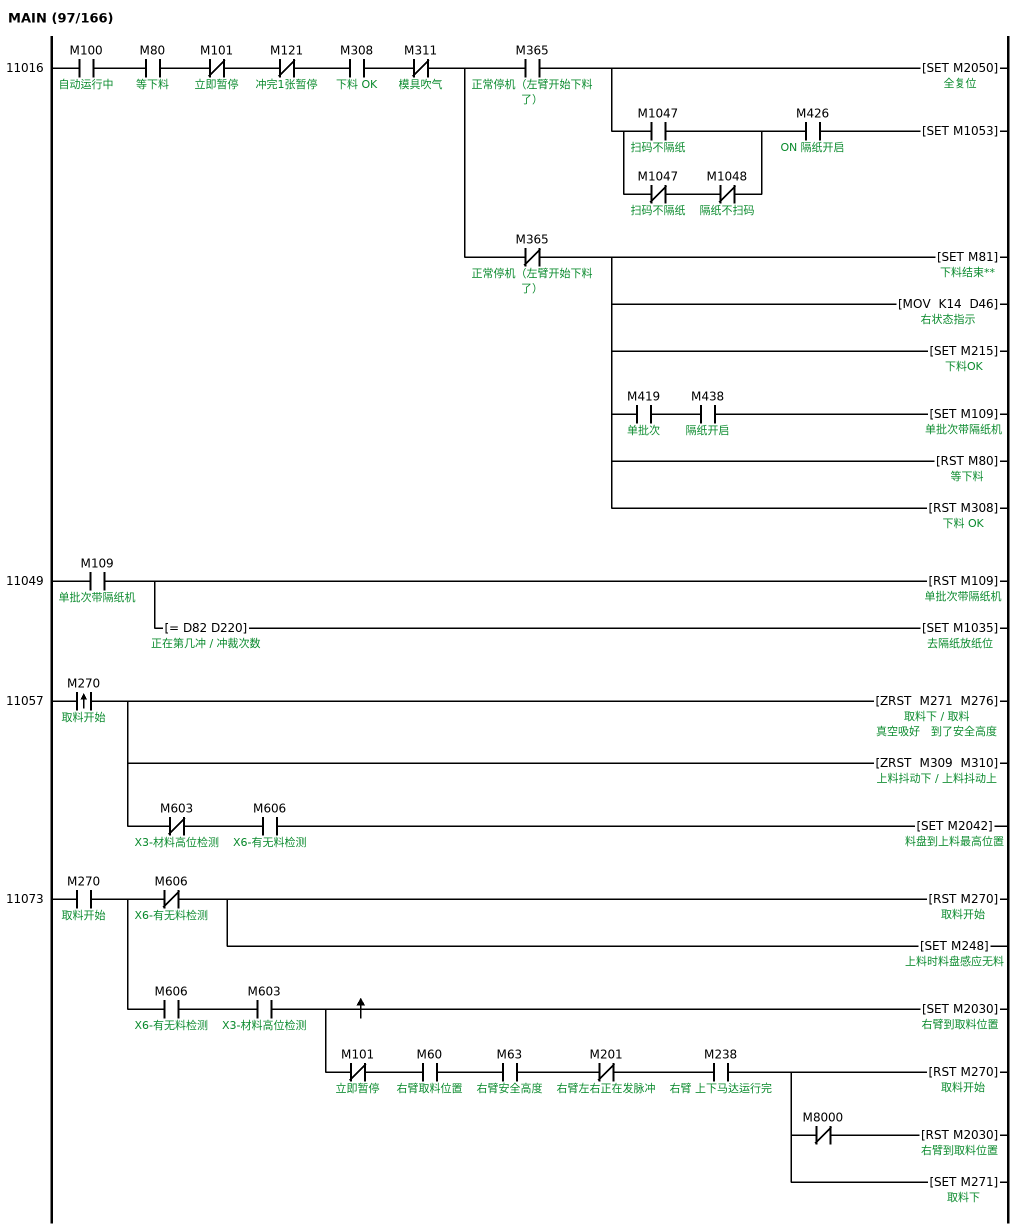
[picture p96: ladder of MAIN, rungs at steps 11016 to 11073]
11016 LD      M100  ; 自动运行中
      AND     M80  ; 等下料
      ANI     M101  ; 立即暂停
      ANI     M121  ; 冲完1张暂停
      AND     M308  ; 下料 OK
      ANI     M311  ; 模具吹气
      MPS
      AND     M365  ; 正常停机（左臂开始下料了）
      SET     M2050  ; 全复位
      LD      M1047  ; 扫码不隔纸
      LDI     M1047  ; 扫码不隔纸
      ANI     M1048  ; 隔纸不扫码
      ORB
      ANB
      AND     M426  ; ON 隔纸开启
      SET     M1053
      MPP
      ANI     M365  ; 正常停机（左臂开始下料了）
      SET     M81  ; 下料结束**
      MOV     K14 D46
      SET     M215  ; 下料OK
      MPS
      AND     M419  ; 单批次
      AND     M438  ; 隔纸开启
      SET     M109  ; 单批次带隔纸机
      MPP
      RST     M80  ; 等下料
      RST     M308  ; 下料 OK
11049 LD      M109  ; 单批次带隔纸机
      RST     M109  ; 单批次带隔纸机
      AND=    D82 D220  ; 正在第几冲 / 冲裁次数
      SET     M1035  ; 去隔纸放纸位
11057 LDP     M270  ; 取料开始
      ZRST    M271 M276  ; 取料下
        [note] M271亮，安全高度不动时，启动此行
      ZRST    M309 M310  ; 上料抖动下 / 上料抖动上
      ANI     M603  ; X3-材料高位检测
      AND     M606  ; X6-有无料检测
      SET     M2042  ; 料盘到上料最高位置
11073 LD      M270  ; 取料开始
      MPS
      ANI     M606  ; X6-有无料检测
      RST     M270  ; 取料开始
      SET     M248  ; 上料时料盘感应无料
      MPP
      AND     M606  ; X6-有无料检测
      AND     M603  ; X3-材料高位检测
      MPS
      MEP
      SET     M2030  ; 右臂到取料位置
      MPP
      ANI     M101  ; 立即暂停
      AND     M60  ; 右臂取料位置
      AND     M63  ; 右臂安全高度
      ANI     M201  ; 右臂左右正在发脉冲
      AND     M238  ; 右臂 上下马达运行完
      RST     M270  ; 取料开始
      MPS
      ANI     M8000
      RST     M2030  ; 右臂到取料位置
      MPP
      SET     M271  ; 取料下
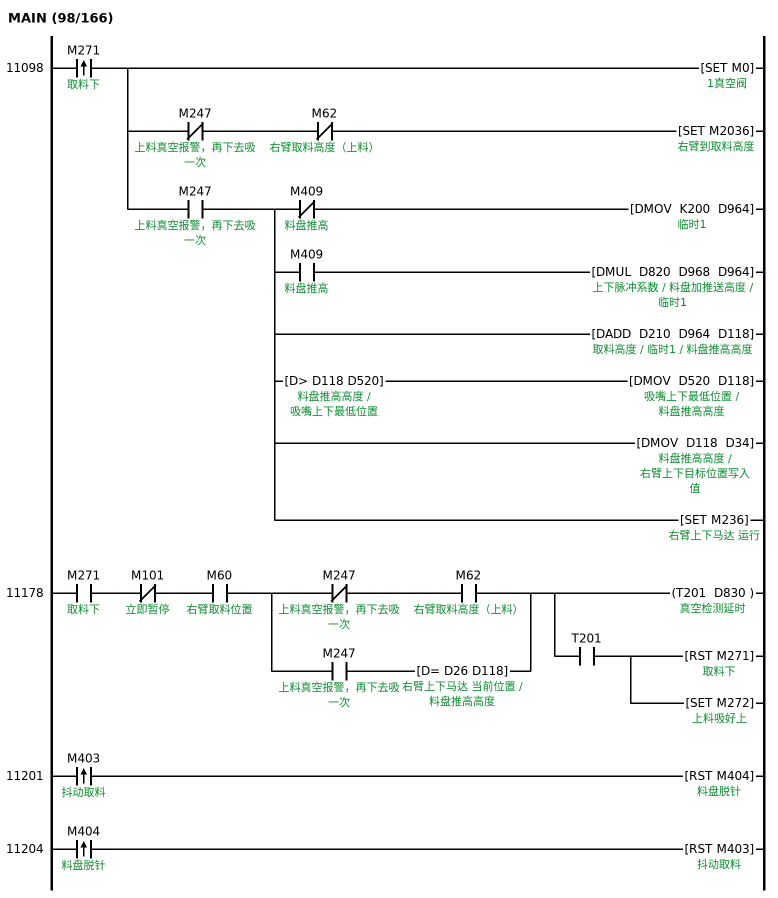
11098 LDP     M271  ; 取料下
      SET     M0  ; 1真空阀
      MPS
      ANI     M247  ; 上料真空报警，再下去吸一次
      ANI     M62  ; 右臂取料高度（上料）
      SET     M2036  ; 右臂到取料高度
      MPP
      AND     M247  ; 上料真空报警，再下去吸一次
      MPS
      ANI     M409  ; 料盘推高
      DMOV    K200 D964
      MRD
      AND     M409  ; 料盘推高
      DMUL    D820 D968 D964
      MPP
      DADD    D210 D964 D118  ; 料盘推高高度
      MPS
      ANDD>   D118 D520  ; 料盘推高高度 / 吸嘴上下最低位置
      DMOV    D520 D118
      MPP
      DMOV    D118 D34
      SET     M236  ; 右臂上下马达 运行
11178 LD      M271  ; 取料下
      ANI     M101  ; 立即暂停
      AND     M60  ; 右臂取料位置
      LDI     M247  ; 上料真空报警，再下去吸一次
      AND     M62  ; 右臂取料高度（上料）
      LD      M247  ; 上料真空报警，再下去吸一次
      ANDD=   D26 D118  ; 右臂上下马达 当前位置 / 料盘推高高度
      ORB
      ANB
      OUT     T201 D830  ; 真空检测延时
      AND     T201
      RST     M271  ; 取料下
      SET     M272  ; 上料吸好上
11201 LDP     M403  ; 抖动取料
      RST     M404  ; 料盘脱针
11204 LDP     M404  ; 料盘脱针
      RST     M403  ; 抖动取料
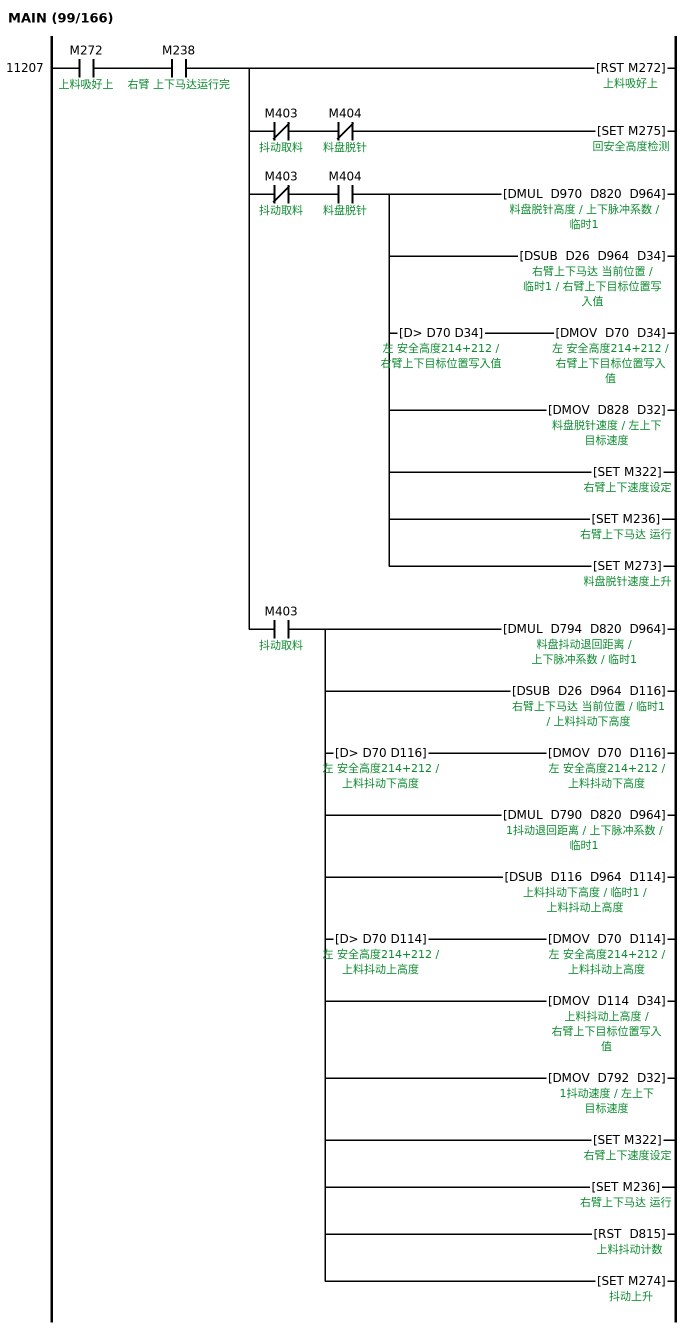
11207 LD      M272  ; 上料吸好上
      AND     M238  ; 右臂 上下马达运行完
      RST     M272  ; 上料吸好上
      MPS
      ANI     M403  ; 抖动取料
      ANI     M404  ; 料盘脱针
      SET     M275  ; 回安全高度检测
      MRD
      ANI     M403  ; 抖动取料
      AND     M404  ; 料盘脱针
      DMUL    D970 D820 D964  ; 料盘脱针高度
      DSUB    D26 D964 D34
      MPS
      ANDD>   D70 D34  ; 左 安全高度214+212 / 右臂上下目标位置写入值
      DMOV    D70 D34
      MPP
      DMOV    D828 D32  ; 左上下 目标速度
      SET     M322  ; 右臂上下速度设定
      SET     M236  ; 右臂上下马达 运行
      SET     M273  ; 料盘脱针速度上升
      MPP
      AND     M403  ; 抖动取料
      DMUL    D794 D820 D964
      DSUB    D26 D964 D116  ; 上料抖动下高度
      MPS
      ANDD>   D70 D116  ; 左 安全高度214+212 / 上料抖动下高度
      DMOV    D70 D116
      MPP
      DMUL    D790 D820 D964
      DSUB    D116 D964 D114  ; 上料抖动上高度
      MPS
      ANDD>   D70 D114  ; 左 安全高度214+212 / 上料抖动上高度
      DMOV    D70 D114
      MPP
      DMOV    D114 D34
      DMOV    D792 D32
      SET     M322  ; 右臂上下速度设定
      SET     M236  ; 右臂上下马达 运行
      RST     D815  ; 上料抖动计数
      SET     M274  ; 抖动上升
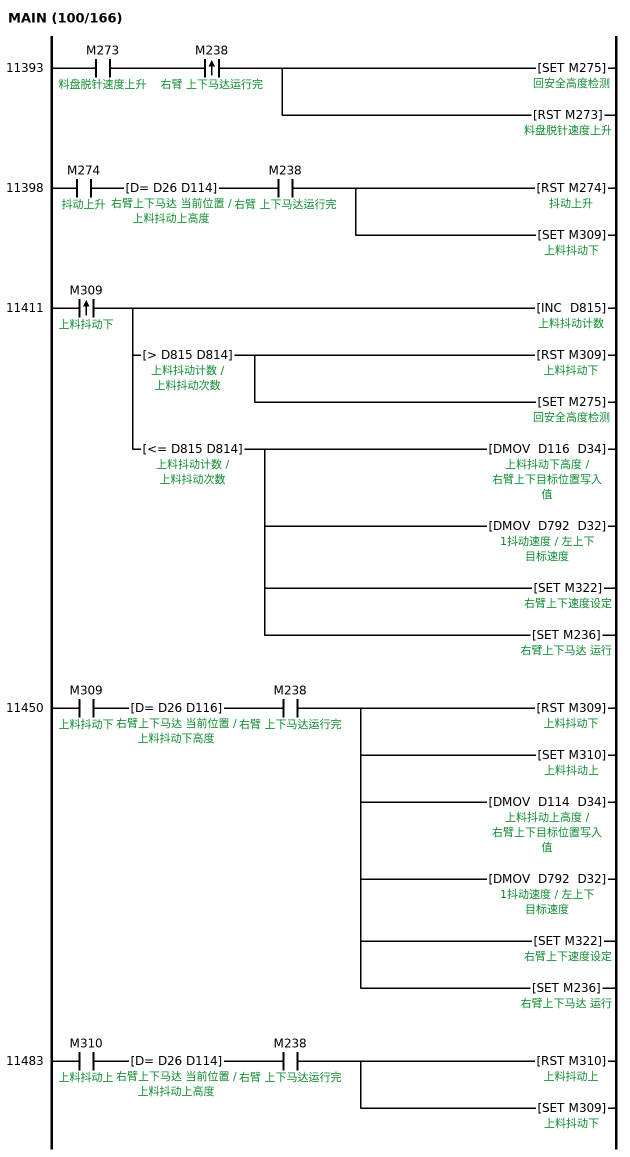
11393 LD      M273  ; 料盘脱针速度上升
      ANDP    M238  ; 右臂 上下马达运行完
      SET     M275  ; 回安全高度检测
      RST     M273  ; 料盘脱针速度上升
11398 LD      M274  ; 抖动上升
      ANDD=   D26 D114  ; 右臂上下马达 当前位置 / 上料抖动上高度
      AND     M238  ; 右臂 上下马达运行完
      RST     M274  ; 抖动上升
      SET     M309  ; 上料抖动下
11411 LDP     M309  ; 上料抖动下
      INC     D815
      MPS
      AND>    D815 D814  ; 上料抖动计数 / 上料抖动次数
      RST     M309  ; 上料抖动下
      SET     M275  ; 回安全高度检测
      MPP
      AND<=   D815 D814  ; 上料抖动计数 / 上料抖动次数
      DMOV    D116 D34
      DMOV    D792 D32
      SET     M322  ; 右臂上下速度设定
      SET     M236  ; 右臂上下马达 运行
11450 LD      M309  ; 上料抖动下
      ANDD=   D26 D116  ; 右臂上下马达 当前位置 / 上料抖动下高度
      AND     M238  ; 右臂 上下马达运行完
      RST     M309  ; 上料抖动下
      SET     M310  ; 上料抖动上
      DMOV    D114 D34
      DMOV    D792 D32
      SET     M322  ; 右臂上下速度设定
      SET     M236  ; 右臂上下马达 运行
11483 LD      M310  ; 上料抖动上
      ANDD=   D26 D114  ; 右臂上下马达 当前位置 / 上料抖动上高度
      AND     M238  ; 右臂 上下马达运行完
      RST     M310  ; 上料抖动上
      SET     M309  ; 上料抖动下
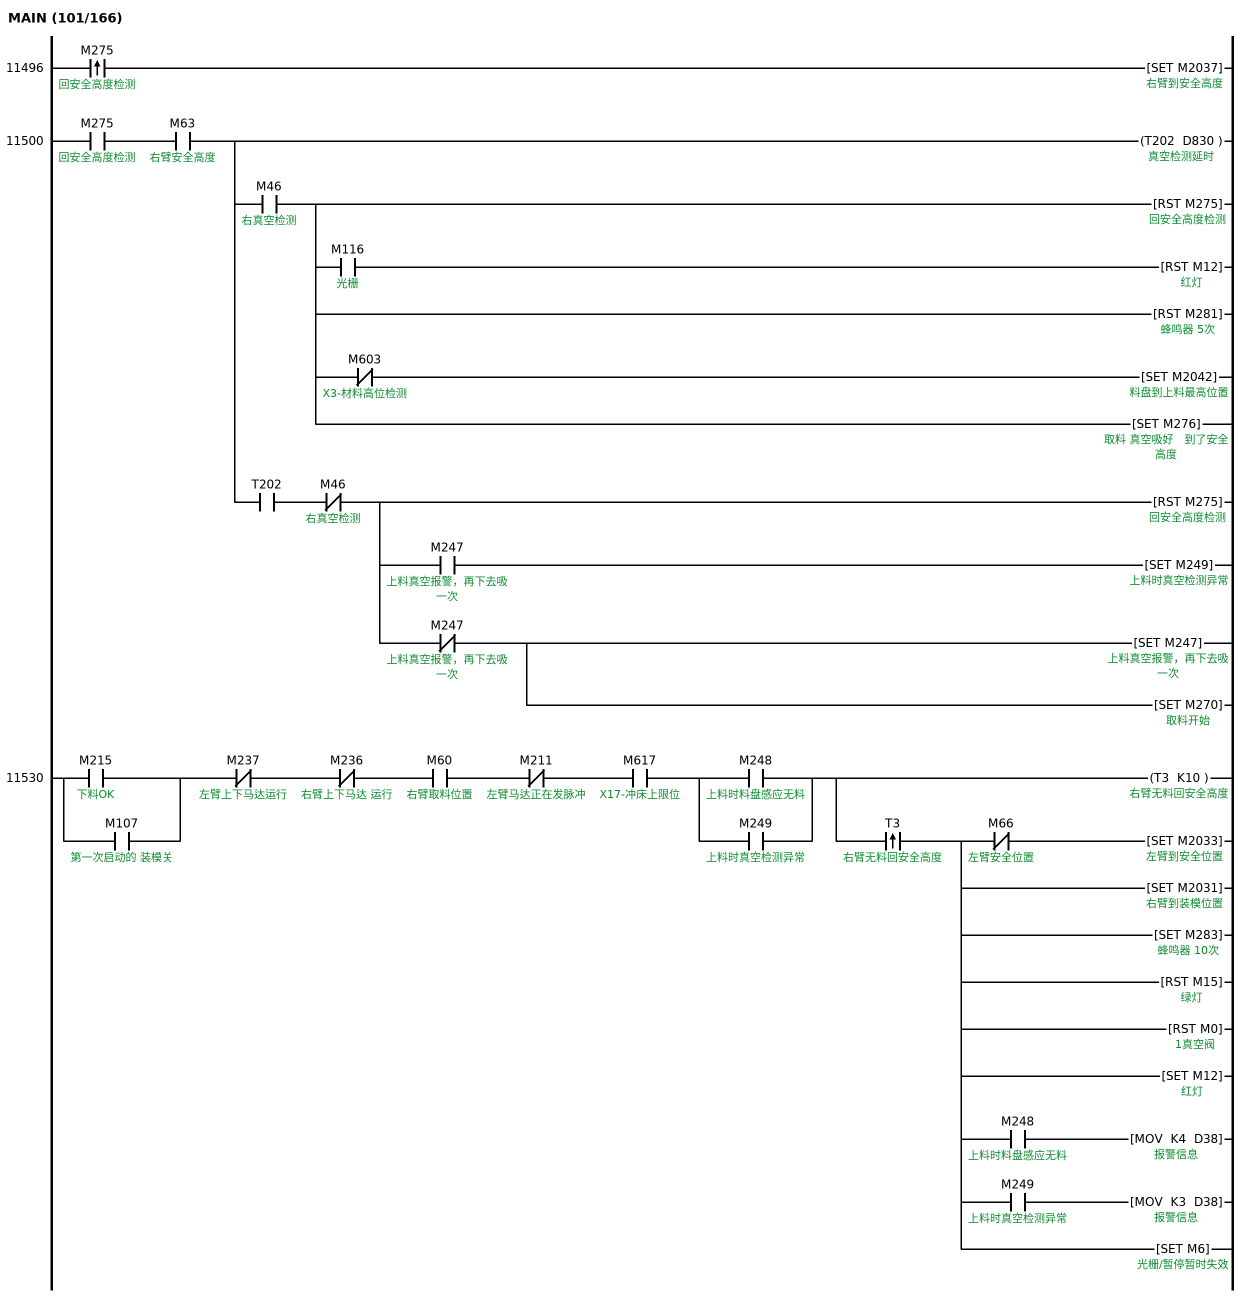
11496 LDP     M275  ; 回安全高度检测
      SET     M2037  ; 右臂到安全高度
11500 LD      M275  ; 回安全高度检测
      AND     M63  ; 右臂安全高度
      OUT     T202 D830  ; 真空检测延时
      MPS
      AND     M46  ; 右真空检测
      RST     M275  ; 回安全高度检测
      MPS
      AND     M116  ; 光栅
      RST     M12  ; 红灯
      MPP
      RST     M281  ; 蜂鸣器 5次
      MPS
      ANI     M603  ; X3-材料高位检测
      SET     M2042  ; 料盘到上料最高位置
      MPP
      SET     M276  ; 取料 真空吸好　到了安全高度
      MPP
      AND     T202
      ANI     M46  ; 右真空检测
      RST     M275  ; 回安全高度检测
      MPS
      AND     M247  ; 上料真空报警，再下去吸一次
      SET     M249  ; 上料时真空检测异常
      MPP
      ANI     M247  ; 上料真空报警，再下去吸一次
      SET     M247  ; 上料真空报警，再下去吸一次
      SET     M270  ; 取料开始
11530 LD      M215  ; 下料OK
      OR      M107  ; 第一次启动的 装模关
      ANI     M237  ; 左臂上下马达运行
      ANI     M236  ; 右臂上下马达 运行
      AND     M60  ; 右臂取料位置
      ANI     M211  ; 左臂马达正在发脉冲
      AND     M617  ; X17-冲床上限位
      LD      M248  ; 上料时料盘感应无料
      OR      M249  ; 上料时真空检测异常
      ANB
      OUT     T3 K10  ; 右臂无料回安全高度
      ANDP    T3  ; 右臂无料回安全高度
      MPS
      ANI     M66  ; 左臂安全位置
      SET     M2033  ; 左臂到安全位置
      MPP
      SET     M2031  ; 右臂到装模位置
      SET     M283  ; 蜂鸣器 10次
      RST     M15  ; 绿灯
      RST     M0  ; 1真空阀
      SET     M12  ; 红灯
      MPS
      AND     M248  ; 上料时料盘感应无料
      MOV     K4 D38
      MRD
      AND     M249  ; 上料时真空检测异常
      MOV     K3 D38
      MPP
      SET     M6  ; 光栅/暂停暂时失效
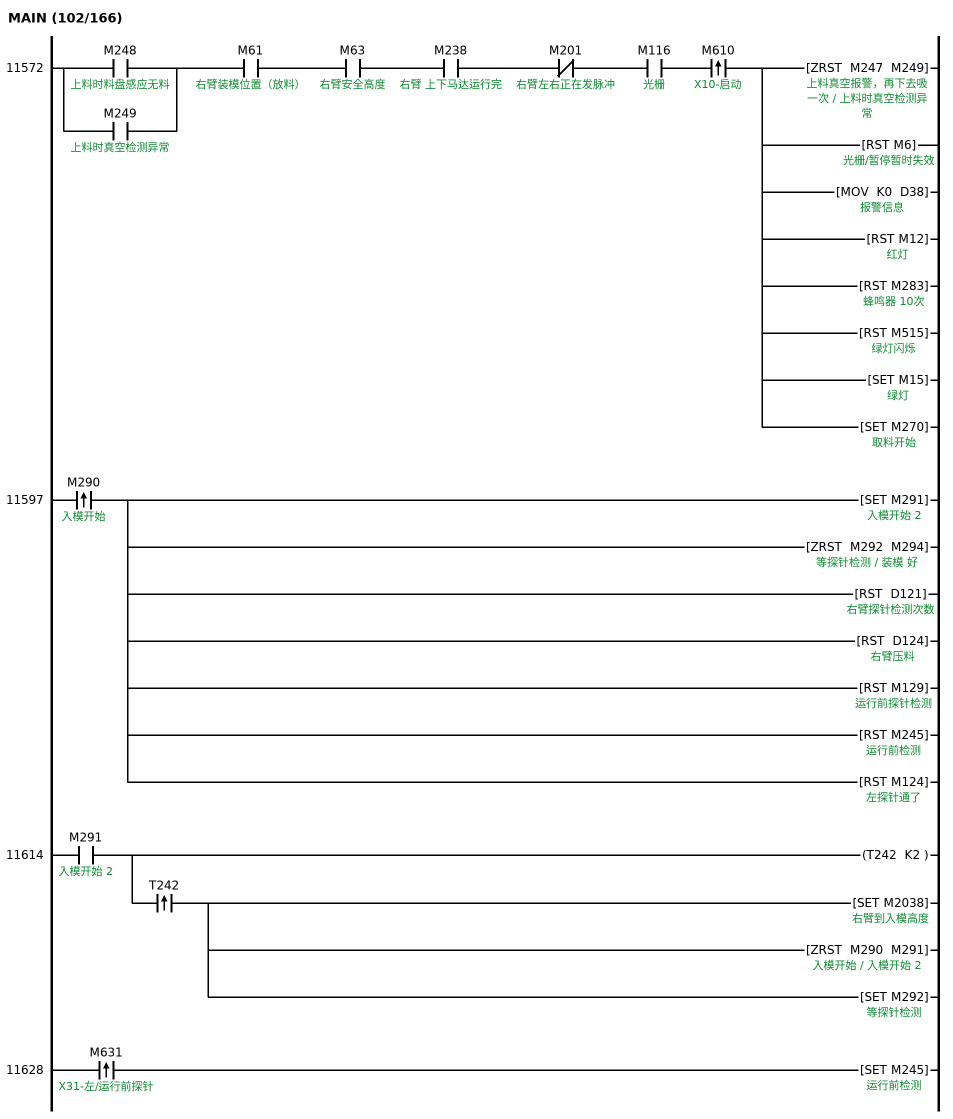
11572 LD      M248  ; 上料时料盘感应无料
      OR      M249  ; 上料时真空检测异常
      AND     M61  ; 右臂装模位置（放料）
      AND     M63  ; 右臂安全高度
      AND     M238  ; 右臂 上下马达运行完
      ANI     M201  ; 右臂左右正在发脉冲
      AND     M116  ; 光栅
      ANDP    M610  ; X10-启动
      ZRST    M247 M249
      RST     M6  ; 光栅/暂停暂时失效
      MOV     K0 D38
      RST     M12  ; 红灯
      RST     M283  ; 蜂鸣器 10次
      RST     M515  ; 绿灯闪烁
      SET     M15  ; 绿灯
      SET     M270  ; 取料开始
11597 LDP     M290  ; 入模开始
      SET     M291  ; 入模开始 2
      ZRST    M292 M294  ; 等探针检测
      RST     D121  ; 右臂探针检测次数
      RST     D124  ; 右臂压料
      RST     M129  ; 运行前探针检测
      RST     M245  ; 运行前检测
      RST     M124  ; 左探针通了
11614 LD      M291  ; 入模开始 2
      OUT     T242 K2
      ANDP    T242
      SET     M2038  ; 右臂到入模高度
      ZRST    M290 M291
      SET     M292  ; 等探针检测
11628 LDP     M631  ; X31-左/运行前探针
      SET     M245  ; 运行前检测
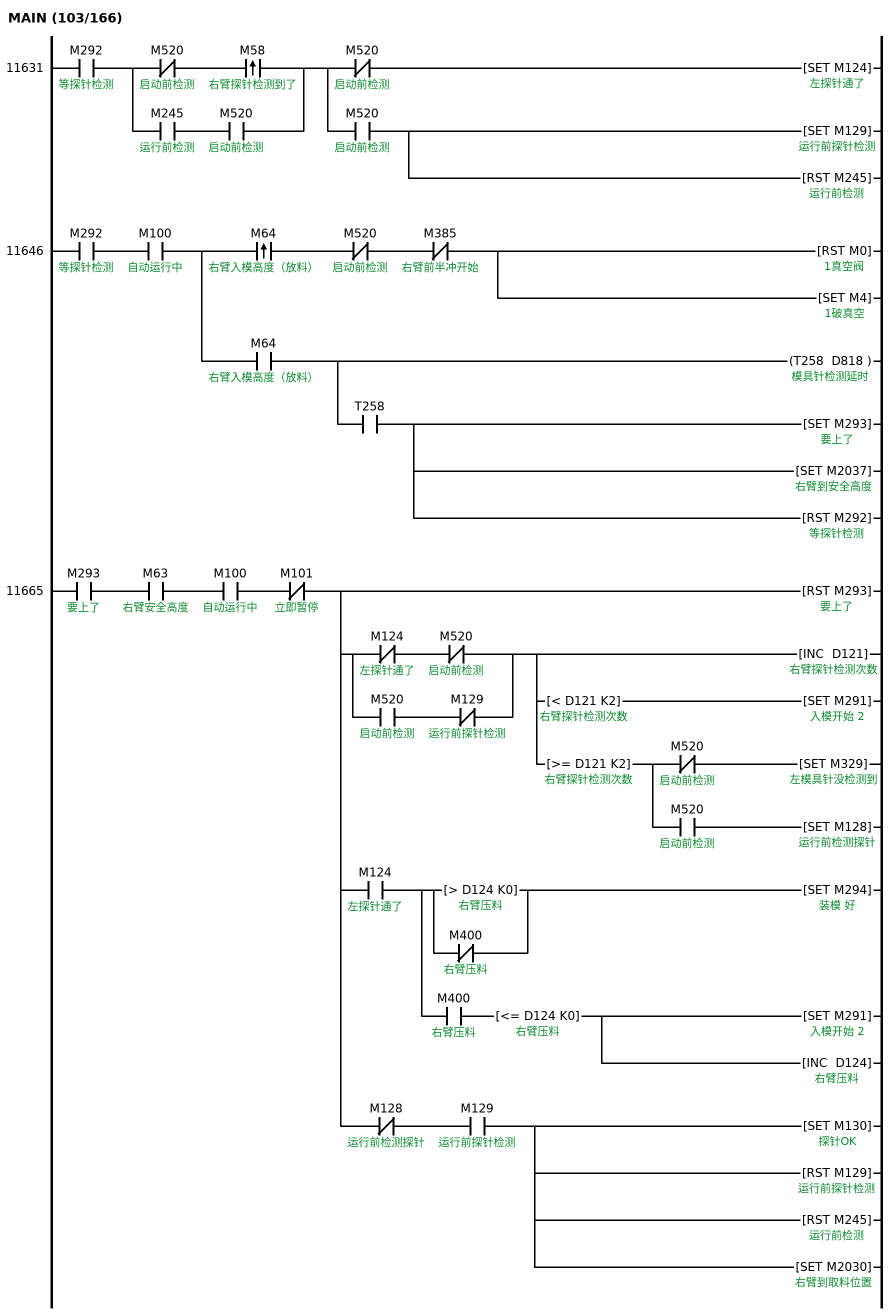
11631 LD      M292  ; 等探针检测
      LDI     M520  ; 启动前检测
      ANDP    M58  ; 右臂探针检测到了
      LD      M245  ; 运行前检测
      AND     M520  ; 启动前检测
      ORB
      ANB
      MPS
      ANI     M520  ; 启动前检测
      SET     M124  ; 左探针通了
      MPP
      AND     M520  ; 启动前检测
      SET     M129  ; 运行前探针检测
      RST     M245  ; 运行前检测
11646 LD      M292  ; 等探针检测
      AND     M100  ; 自动运行中
      MPS
      ANDP    M64  ; 右臂入模高度（放料）
      ANI     M520  ; 启动前检测
      ANI     M385  ; 右臂前半冲开始
      RST     M0  ; 1真空阀
      SET     M4  ; 1破真空
      MPP
      AND     M64  ; 右臂入模高度（放料）
      OUT     T258 D818  ; 模具针检测延时
      AND     T258
      SET     M293  ; 要上了
      SET     M2037  ; 右臂到安全高度
      RST     M292  ; 等探针检测
11665 LD      M293  ; 要上了
      AND     M63  ; 右臂安全高度
      AND     M100  ; 自动运行中
      ANI     M101  ; 立即暂停
      RST     M293  ; 要上了
      MPS
      LDI     M124  ; 左探针通了
      ANI     M520  ; 启动前检测
      LD      M520  ; 启动前检测
      ANI     M129  ; 运行前探针检测
      ORB
      ANB
      INC     D121
      MPS
      AND<    D121 K2  ; 右臂探针检测次数
      SET     M291  ; 入模开始 2
      MPP
      AND>=   D121 K2  ; 右臂探针检测次数
      MPS
      ANI     M520  ; 启动前检测
      SET     M329  ; 左模具针没检测到
      MPP
      AND     M520  ; 启动前检测
      SET     M128  ; 运行前检测探针
      MRD
      AND     M124  ; 左探针通了
      MPS
      LD>     D124 K0  ; 右臂压料
      ORI     M400  ; 右臂压料
      ANB
      SET     M294  ; 装模 好
      MPP
      AND     M400  ; 右臂压料
      AND<=   D124 K0  ; 右臂压料
      SET     M291  ; 入模开始 2
      INC     D124
      MPP
      ANI     M128  ; 运行前检测探针
      AND     M129  ; 运行前探针检测
      SET     M130  ; 探针OK
      RST     M129  ; 运行前探针检测
      RST     M245  ; 运行前检测
      SET     M2030  ; 右臂到取料位置
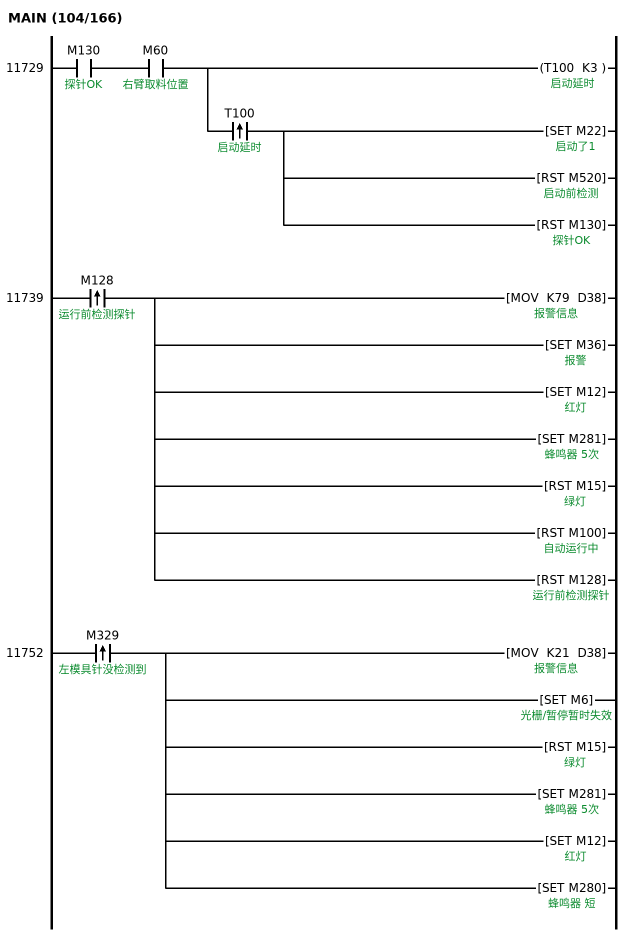
11729 LD      M130  ; 探针OK
      AND     M60  ; 右臂取料位置
      OUT     T100 K3  ; 启动延时
      ANDP    T100  ; 启动延时
      SET     M22  ; 启动了1
      RST     M520  ; 启动前检测
      RST     M130  ; 探针OK
11739 LDP     M128  ; 运行前检测探针
      MOV     K79 D38
      SET     M36  ; 报警
      SET     M12  ; 红灯
      SET     M281  ; 蜂鸣器 5次
      RST     M15  ; 绿灯
      RST     M100  ; 自动运行中
      RST     M128  ; 运行前检测探针
11752 LDP     M329  ; 左模具针没检测到
      MOV     K21 D38
      SET     M6  ; 光栅/暂停暂时失效
      RST     M15  ; 绿灯
      SET     M281  ; 蜂鸣器 5次
      SET     M12  ; 红灯
      SET     M280  ; 蜂鸣器 短
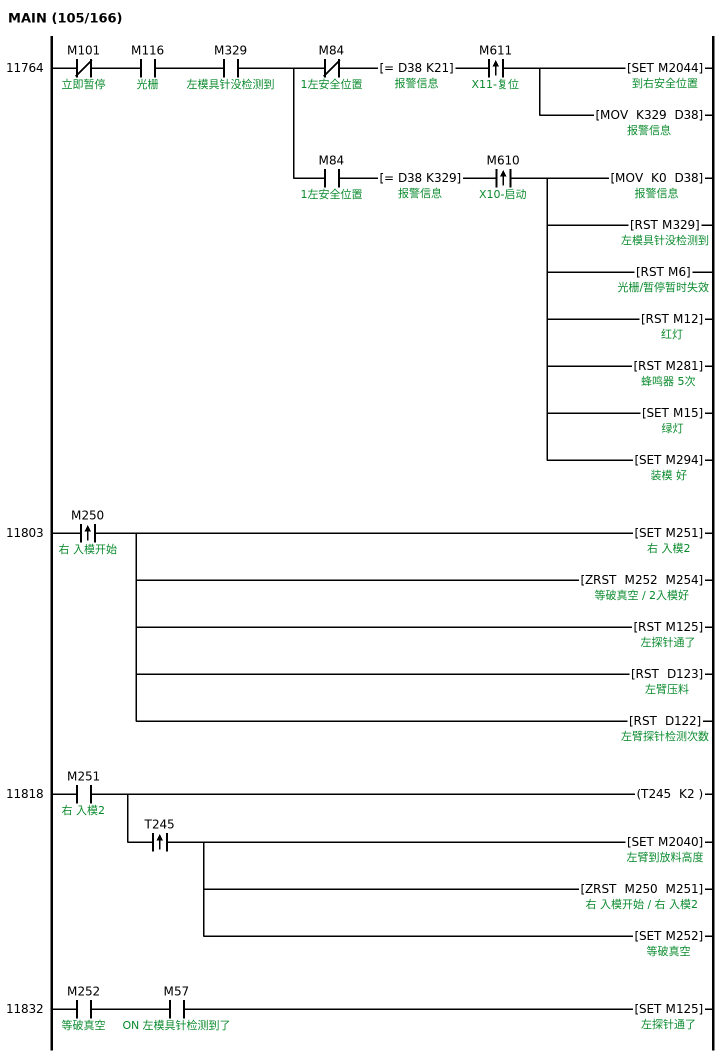
11764 LDI     M101  ; 立即暂停
      AND     M116  ; 光栅
      AND     M329  ; 左模具针没检测到
      MPS
      ANI     M84  ; 1左安全位置
      AND=    D38 K21  ; 报警信息
      ANDP    M611  ; X11-复位
      SET     M2044  ; 到右安全位置
      MOV     K329 D38
      MPP
      AND     M84  ; 1左安全位置
      AND=    D38 K329  ; 报警信息
      ANDP    M610  ; X10-启动
      MOV     K0 D38
      RST     M329  ; 左模具针没检测到
      RST     M6  ; 光栅/暂停暂时失效
      RST     M12  ; 红灯
      RST     M281  ; 蜂鸣器 5次
      SET     M15  ; 绿灯
      SET     M294  ; 装模 好
11803 LDP     M250  ; 右 入模开始
      SET     M251  ; 右 入模2
      ZRST    M252 M254  ; 等破真空
      RST     M125  ; 左探针通了
      RST     D123  ; 左臂压料
      RST     D122  ; 左臂探针检测次数
11818 LD      M251  ; 右 入模2
      OUT     T245 K2
      ANDP    T245
      SET     M2040  ; 左臂到放料高度
      ZRST    M250 M251
      SET     M252  ; 等破真空
11832 LD      M252  ; 等破真空
      AND     M57  ; ON 左模具针检测到了
      SET     M125  ; 左探针通了
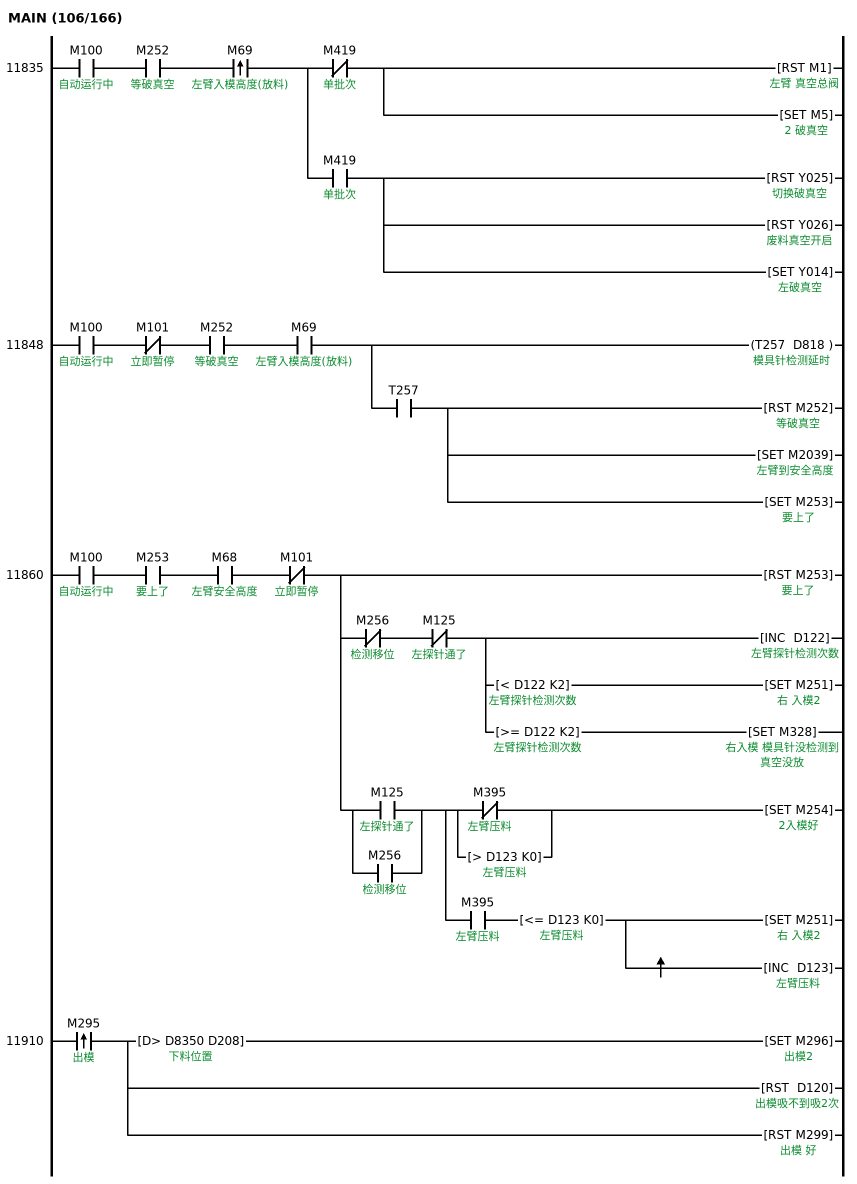
11835 LD      M100  ; 自动运行中
      AND     M252  ; 等破真空
      ANDP    M69  ; 左臂入模高度(放料)
      MPS
      ANI     M419  ; 单批次
      RST     M1  ; 左臂 真空总阀
      SET     M5  ; 2 破真空
      MPP
      AND     M419  ; 单批次
      RST     Y025  ; 切换破真空
      RST     Y026  ; 废料真空开启
      SET     Y014  ; 左破真空
11848 LD      M100  ; 自动运行中
      ANI     M101  ; 立即暂停
      AND     M252  ; 等破真空
      AND     M69  ; 左臂入模高度(放料)
      OUT     T257 D818  ; 模具针检测延时
      AND     T257
      RST     M252  ; 等破真空
      SET     M2039  ; 左臂到安全高度
      SET     M253  ; 要上了
11860 LD      M100  ; 自动运行中
      AND     M253  ; 要上了
      AND     M68  ; 左臂安全高度
      ANI     M101  ; 立即暂停
      RST     M253  ; 要上了
      MPS
      ANI     M256  ; 检测移位
      ANI     M125  ; 左探针通了
      INC     D122
      MPS
      AND<    D122 K2  ; 左臂探针检测次数
      SET     M251  ; 右 入模2
      MPP
      AND>=   D122 K2  ; 左臂探针检测次数
      SET     M328  ; 右入模 模具针没检测到 真空没放
      MPP
      LD      M125  ; 左探针通了
      OR      M256  ; 检测移位
      ANB
      MPS
      LDI     M395  ; 左臂压料
      OR>     D123 K0  ; 左臂压料
      ANB
      SET     M254  ; 2入模好
      MPP
      AND     M395  ; 左臂压料
      AND<=   D123 K0  ; 左臂压料
      SET     M251  ; 右 入模2
      MEP
      INC     D123
11910 LDP     M295  ; 出模
      MPS
      ANDD>   D8350 D208  ; 下料位置
      SET     M296  ; 出模2
      MPP
      RST     D120  ; 出模吸不到吸2次
      RST     M299  ; 出模 好
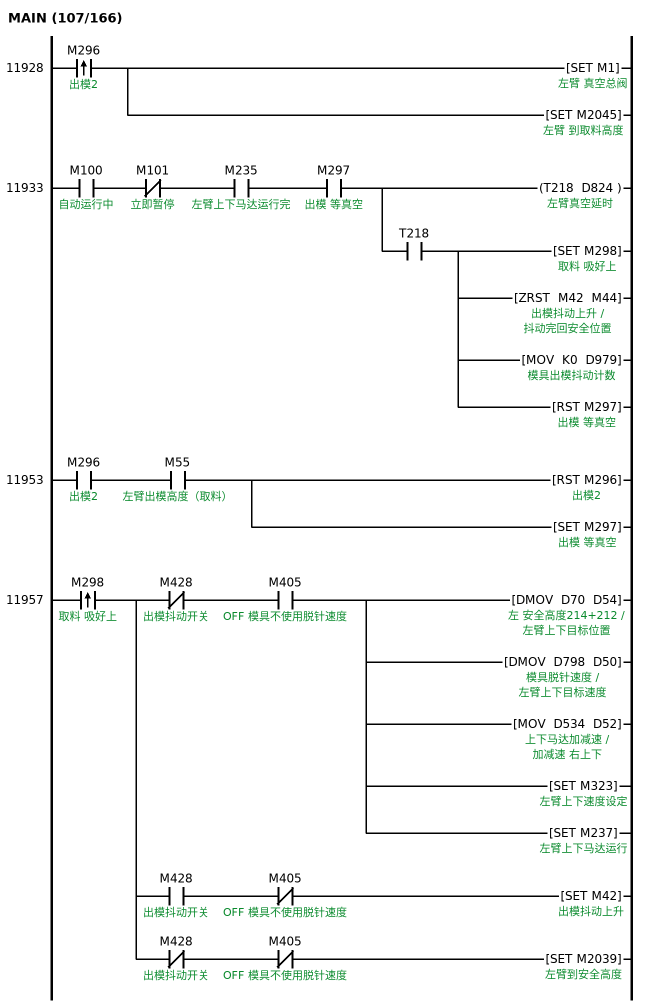
11928 LDP     M296  ; 出模2
      SET     M1  ; 左臂 真空总阀
      SET     M2045  ; 左臂 到取料高度
11933 LD      M100  ; 自动运行中
      ANI     M101  ; 立即暂停
      AND     M235  ; 左臂上下马达运行完
      AND     M297  ; 出模 等真空
      OUT     T218 D824  ; 左臂真空延时
      AND     T218
      SET     M298  ; 取料 吸好上
      ZRST    M42 M44  ; 出模抖动上升 / 抖动完回安全位置
      MOV     K0 D979  ; 模具出模抖动计数
      RST     M297  ; 出模 等真空
11953 LD      M296  ; 出模2
      AND     M55  ; 左臂出模高度（取料）
      RST     M296  ; 出模2
      SET     M297  ; 出模 等真空
11957 LDP     M298  ; 取料 吸好上
      MPS
      ANI     M428  ; 出模抖动开关
      AND     M405  ; OFF 模具不使用脱针速度
      DMOV    D70 D54  ; 左臂上下目标位置
      DMOV    D798 D50  ; 左臂上下目标速度
      MOV     D534 D52  ; 加减速 右上下
      SET     M323  ; 左臂上下速度设定
      SET     M237  ; 左臂上下马达运行
      MRD
      AND     M428  ; 出模抖动开关
      ANI     M405  ; OFF 模具不使用脱针速度
      SET     M42  ; 出模抖动上升
      MPP
      ANI     M428  ; 出模抖动开关
      ANI     M405  ; OFF 模具不使用脱针速度
      SET     M2039  ; 左臂到安全高度
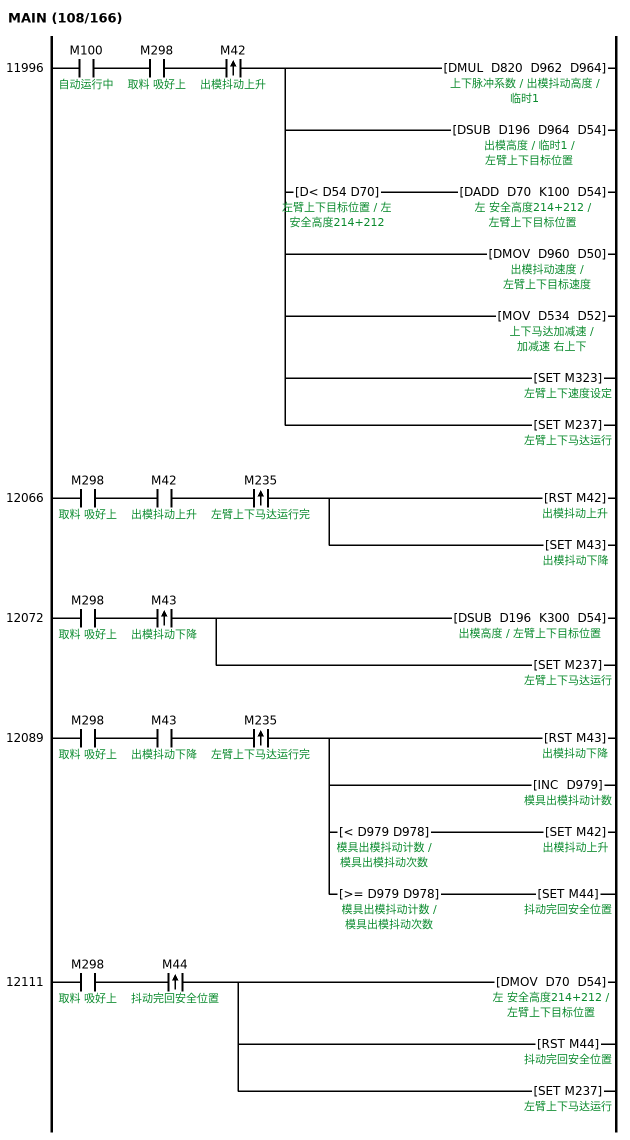
11996 LD      M100  ; 自动运行中
      AND     M298  ; 取料 吸好上
      ANDP    M42  ; 出模抖动上升
      DMUL    D820 D962 D964
      DSUB    D196 D964 D54
      MPS
      ANDD<   D54 D70  ; 左臂上下目标位置 / 左 安全高度214+212
      DADD    D70 K100 D54
      MPP
      DMOV    D960 D50
      MOV     D534 D52
      SET     M323  ; 左臂上下速度设定
      SET     M237  ; 左臂上下马达运行
12066 LD      M298  ; 取料 吸好上
      AND     M42  ; 出模抖动上升
      ANDP    M235  ; 左臂上下马达运行完
      RST     M42  ; 出模抖动上升
      SET     M43  ; 出模抖动下降
12072 LD      M298  ; 取料 吸好上
      ANDP    M43  ; 出模抖动下降
      DSUB    D196 K300 D54
      SET     M237  ; 左臂上下马达运行
12089 LD      M298  ; 取料 吸好上
      AND     M43  ; 出模抖动下降
      ANDP    M235  ; 左臂上下马达运行完
      RST     M43  ; 出模抖动下降
      INC     D979
      MPS
      AND<    D979 D978  ; 模具出模抖动计数 / 模具出模抖动次数
      SET     M42  ; 出模抖动上升
      MPP
      AND>=   D979 D978  ; 模具出模抖动计数 / 模具出模抖动次数
      SET     M44  ; 抖动完回安全位置
12111 LD      M298  ; 取料 吸好上
      ANDP    M44  ; 抖动完回安全位置
      DMOV    D70 D54
      RST     M44  ; 抖动完回安全位置
      SET     M237  ; 左臂上下马达运行
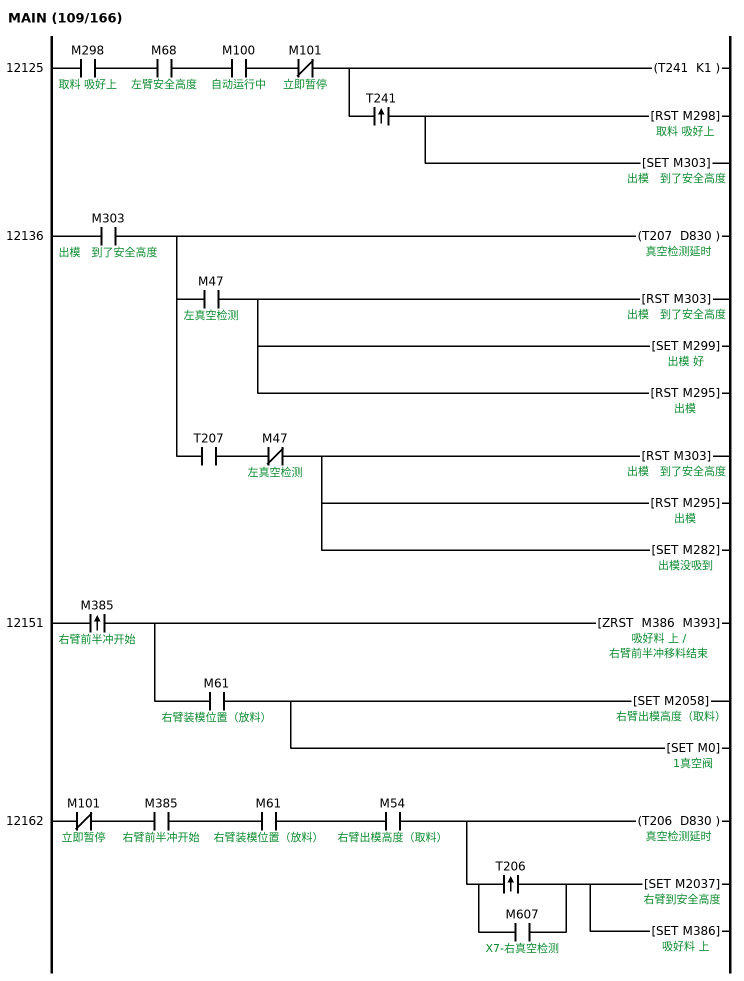
12125 LD      M298  ; 取料 吸好上
      AND     M68  ; 左臂安全高度
      AND     M100  ; 自动运行中
      ANI     M101  ; 立即暂停
      OUT     T241 K1
      ANDP    T241
      RST     M298  ; 取料 吸好上
      SET     M303  ; 出模　到了安全高度
12136 LD      M303  ; 出模　到了安全高度
      OUT     T207 D830  ; 真空检测延时
      MPS
      AND     M47  ; 左真空检测
      RST     M303  ; 出模　到了安全高度
      SET     M299  ; 出模 好
      RST     M295  ; 出模
      MPP
      AND     T207
      ANI     M47  ; 左真空检测
      RST     M303  ; 出模　到了安全高度
      RST     M295  ; 出模
      SET     M282  ; 出模没吸到
12151 LDP     M385  ; 右臂前半冲开始
      ZRST    M386 M393  ; 吸好料 上
      AND     M61  ; 右臂装模位置（放料）
      SET     M2058  ; 右臂出模高度（取料）
      SET     M0  ; 1真空阀
12162 LDI     M101  ; 立即暂停
      AND     M385  ; 右臂前半冲开始
      AND     M61  ; 右臂装模位置（放料）
      AND     M54  ; 右臂出模高度（取料）
      OUT     T206 D830  ; 真空检测延时
      LDP     T206
      OR      M607  ; X7-右真空检测
      ANB
      SET     M2037  ; 右臂到安全高度
      SET     M386  ; 吸好料 上
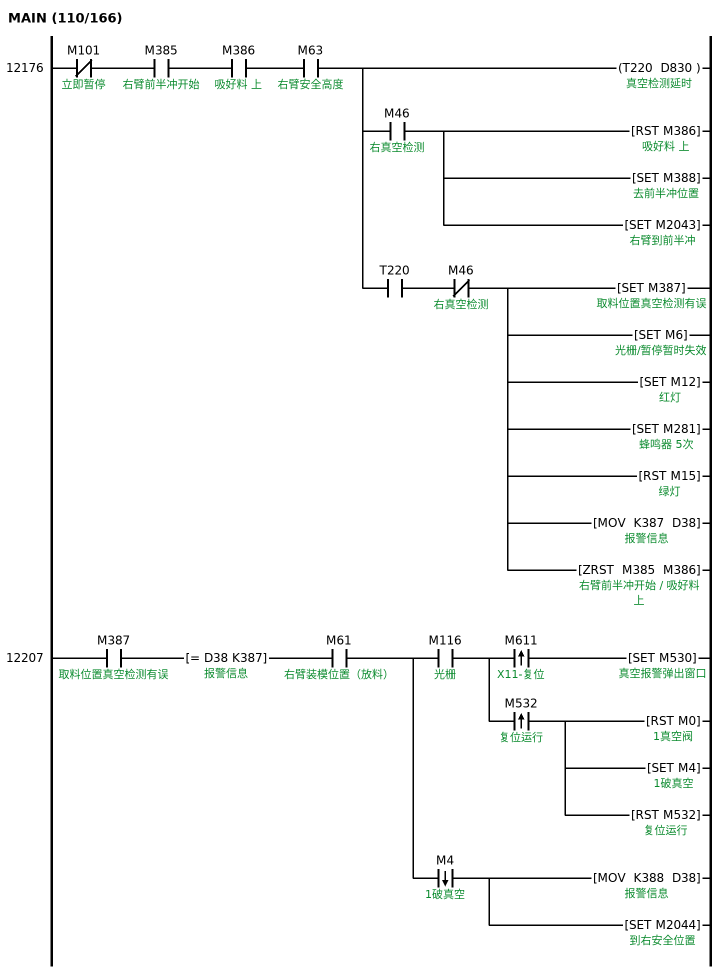
12176 LDI     M101  ; 立即暂停
      AND     M385  ; 右臂前半冲开始
      AND     M386  ; 吸好料 上
      AND     M63  ; 右臂安全高度
      OUT     T220 D830  ; 真空检测延时
      MPS
      AND     M46  ; 右真空检测
      RST     M386  ; 吸好料 上
      SET     M388  ; 去前半冲位置
      SET     M2043  ; 右臂到前半冲
      MPP
      AND     T220
      ANI     M46  ; 右真空检测
      SET     M387  ; 取料位置真空检测有误
      SET     M6  ; 光栅/暂停暂时失效
      SET     M12  ; 红灯
      SET     M281  ; 蜂鸣器 5次
      RST     M15  ; 绿灯
      MOV     K387 D38
      ZRST    M385 M386
12207 LD      M387  ; 取料位置真空检测有误
      AND=    D38 K387  ; 报警信息
      AND     M61  ; 右臂装模位置（放料）
      MPS
      AND     M116  ; 光栅
      MPS
      ANDP    M611  ; X11-复位
      SET     M530  ; 真空报警弹出窗口
      MPP
      ANDP    M532  ; 复位运行
      RST     M0  ; 1真空阀
      SET     M4  ; 1破真空
      RST     M532  ; 复位运行
      MPP
      ANDF    M4  ; 1破真空
      MOV     K388 D38
      SET     M2044  ; 到右安全位置
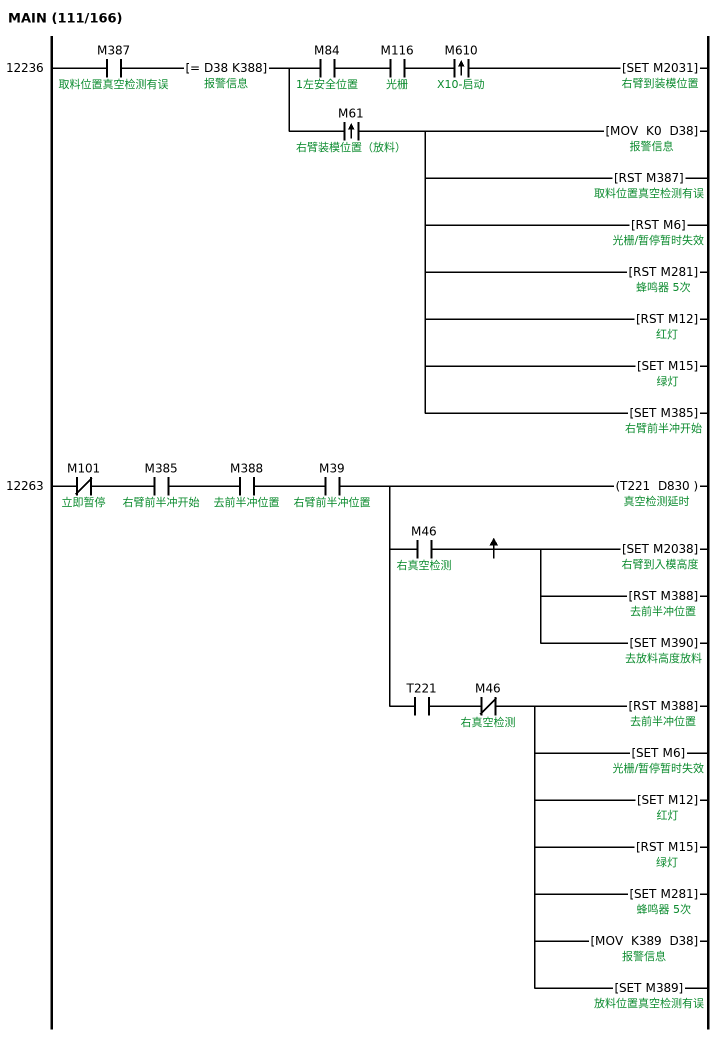
12236 LD      M387  ; 取料位置真空检测有误
      AND=    D38 K388  ; 报警信息
      MPS
      AND     M84  ; 1左安全位置
      AND     M116  ; 光栅
      ANDP    M610  ; X10-启动
      SET     M2031  ; 右臂到装模位置
      MPP
      ANDP    M61  ; 右臂装模位置（放料）
      MOV     K0 D38
      RST     M387  ; 取料位置真空检测有误
      RST     M6  ; 光栅/暂停暂时失效
      RST     M281  ; 蜂鸣器 5次
      RST     M12  ; 红灯
      SET     M15  ; 绿灯
      SET     M385  ; 右臂前半冲开始
12263 LDI     M101  ; 立即暂停
      AND     M385  ; 右臂前半冲开始
      AND     M388  ; 去前半冲位置
      AND     M39  ; 右臂前半冲位置
      OUT     T221 D830  ; 真空检测延时
      MPS
      AND     M46  ; 右真空检测
      MEP
      SET     M2038  ; 右臂到入模高度
      RST     M388  ; 去前半冲位置
      SET     M390  ; 去放料高度放料
      MPP
      AND     T221
      ANI     M46  ; 右真空检测
      RST     M388  ; 去前半冲位置
      SET     M6  ; 光栅/暂停暂时失效
      SET     M12  ; 红灯
      RST     M15  ; 绿灯
      SET     M281  ; 蜂鸣器 5次
      MOV     K389 D38
      SET     M389  ; 放料位置真空检测有误
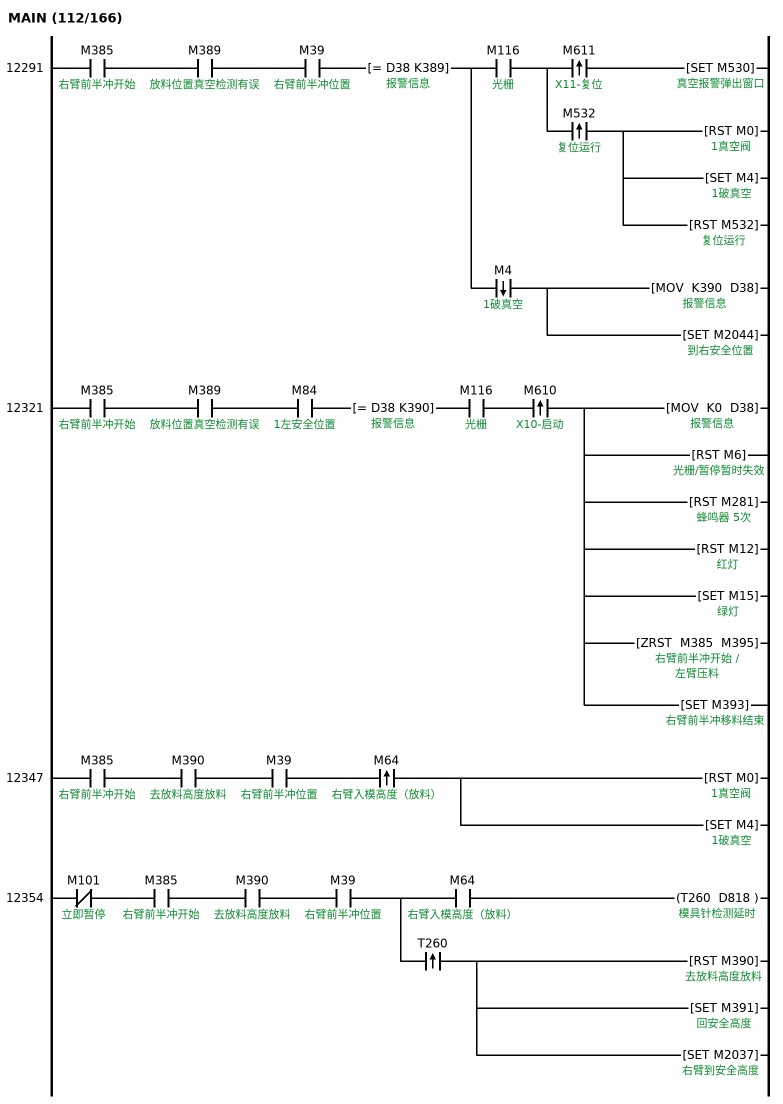
12291 LD      M385  ; 右臂前半冲开始
      AND     M389  ; 放料位置真空检测有误
      AND     M39  ; 右臂前半冲位置
      AND=    D38 K389  ; 报警信息
      MPS
      AND     M116  ; 光栅
      MPS
      ANDP    M611  ; X11-复位
      SET     M530  ; 真空报警弹出窗口
      MPP
      ANDP    M532  ; 复位运行
      RST     M0  ; 1真空阀
      SET     M4  ; 1破真空
      RST     M532  ; 复位运行
      MPP
      ANDF    M4  ; 1破真空
      MOV     K390 D38
      SET     M2044  ; 到右安全位置
12321 LD      M385  ; 右臂前半冲开始
      AND     M389  ; 放料位置真空检测有误
      AND     M84  ; 1左安全位置
      AND=    D38 K390  ; 报警信息
      AND     M116  ; 光栅
      ANDP    M610  ; X10-启动
      MOV     K0 D38
      RST     M6  ; 光栅/暂停暂时失效
      RST     M281  ; 蜂鸣器 5次
      RST     M12  ; 红灯
      SET     M15  ; 绿灯
      ZRST    M385 M395
      SET     M393  ; 右臂前半冲移料结束
12347 LD      M385  ; 右臂前半冲开始
      AND     M390  ; 去放料高度放料
      AND     M39  ; 右臂前半冲位置
      ANDP    M64  ; 右臂入模高度（放料）
      RST     M0  ; 1真空阀
      SET     M4  ; 1破真空
12354 LDI     M101  ; 立即暂停
      AND     M385  ; 右臂前半冲开始
      AND     M390  ; 去放料高度放料
      AND     M39  ; 右臂前半冲位置
      MPS
      AND     M64  ; 右臂入模高度（放料）
      OUT     T260 D818  ; 模具针检测延时
      MPP
      ANDP    T260
      RST     M390  ; 去放料高度放料
      SET     M391  ; 回安全高度
      SET     M2037  ; 右臂到安全高度
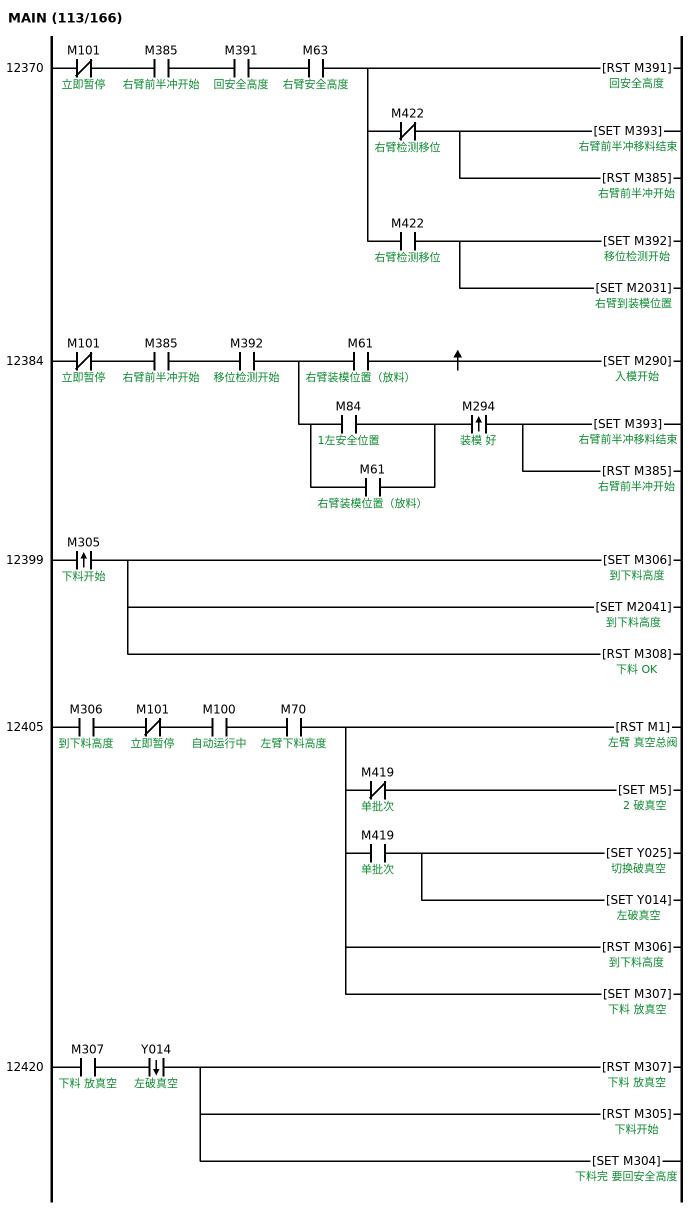
12370 LDI     M101  ; 立即暂停
      AND     M385  ; 右臂前半冲开始
      AND     M391  ; 回安全高度
      AND     M63  ; 右臂安全高度
      RST     M391  ; 回安全高度
      MPS
      ANI     M422  ; 右臂检测移位
      SET     M393  ; 右臂前半冲移料结束
      RST     M385  ; 右臂前半冲开始
      MPP
      AND     M422  ; 右臂检测移位
      SET     M392  ; 移位检测开始
      SET     M2031  ; 右臂到装模位置
12384 LDI     M101  ; 立即暂停
      AND     M385  ; 右臂前半冲开始
      AND     M392  ; 移位检测开始
      MPS
      AND     M61  ; 右臂装模位置（放料）
      MEP
      SET     M290  ; 入模开始
      MPP
      LD      M84  ; 1左安全位置
      OR      M61  ; 右臂装模位置（放料）
      ANB
      ANDP    M294  ; 装模 好
      SET     M393  ; 右臂前半冲移料结束
      RST     M385  ; 右臂前半冲开始
12399 LDP     M305  ; 下料开始
      SET     M306  ; 到下料高度
      SET     M2041  ; 到下料高度
      RST     M308  ; 下料 OK
12405 LD      M306  ; 到下料高度
      ANI     M101  ; 立即暂停
      AND     M100  ; 自动运行中
      AND     M70  ; 左臂下料高度
      RST     M1  ; 左臂 真空总阀
      MPS
      ANI     M419  ; 单批次
      SET     M5  ; 2 破真空
      MRD
      AND     M419  ; 单批次
      SET     Y025  ; 切换破真空
      SET     Y014  ; 左破真空
      MPP
      RST     M306  ; 到下料高度
      SET     M307  ; 下料 放真空
12420 LD      M307  ; 下料 放真空
      ANDF    Y014  ; 左破真空
      RST     M307  ; 下料 放真空
      RST     M305  ; 下料开始
      SET     M304  ; 下料完 要回安全高度
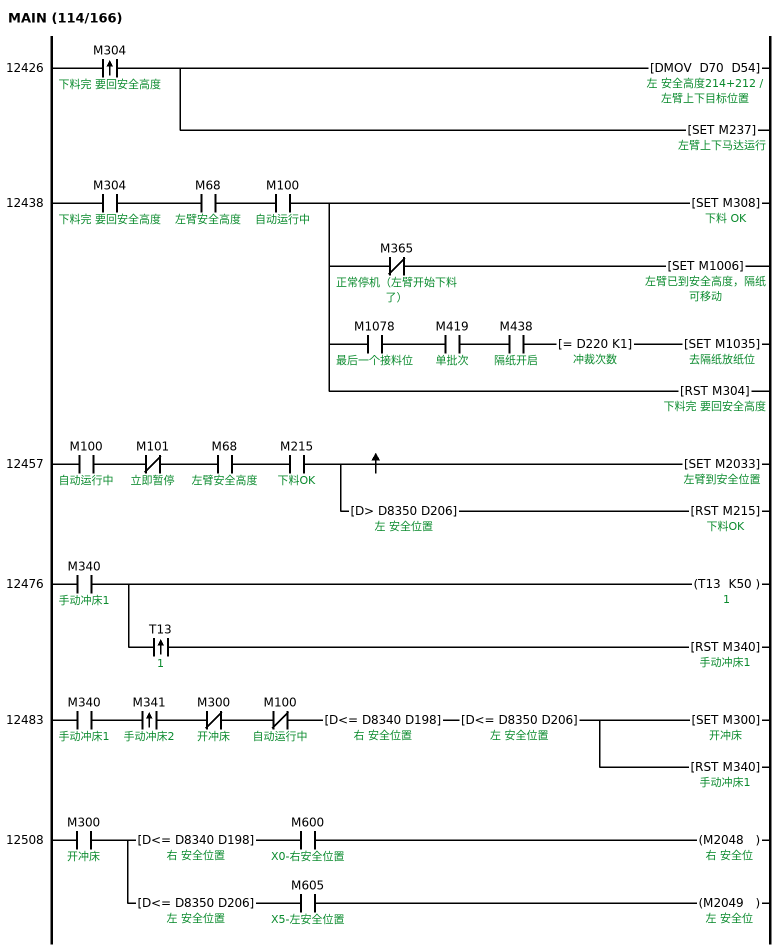
12426 LDP     M304  ; 下料完 要回安全高度
      DMOV    D70 D54
      SET     M237  ; 左臂上下马达运行
12438 LD      M304  ; 下料完 要回安全高度
      AND     M68  ; 左臂安全高度
      AND     M100  ; 自动运行中
      SET     M308  ; 下料 OK
      MPS
      ANI     M365  ; 正常停机（左臂开始下料了）
      SET     M1006  ; 左臂已到安全高度，隔纸可移动
      MRD
      AND     M1078  ; 最后一个接料位
      AND     M419  ; 单批次
      AND     M438  ; 隔纸开启
      AND=    D220 K1  ; 冲裁次数
      SET     M1035  ; 去隔纸放纸位
      MPP
      RST     M304  ; 下料完 要回安全高度
12457 LD      M100  ; 自动运行中
      ANI     M101  ; 立即暂停
      AND     M68  ; 左臂安全高度
      AND     M215  ; 下料OK
      MPS
      MEP
      SET     M2033  ; 左臂到安全位置
      MPP
      ANDD>   D8350 D206  ; 左 安全位置
      RST     M215  ; 下料OK
12476 LD      M340  ; 手动冲床1
      OUT     T13 K50  ; 1
      ANDP    T13  ; 1
      RST     M340  ; 手动冲床1
12483 LD      M340  ; 手动冲床1
      ANDP    M341  ; 手动冲床2
      ANI     M300  ; 开冲床
      ANI     M100  ; 自动运行中
      ANDD<=  D8340 D198  ; 右 安全位置
      ANDD<=  D8350 D206  ; 左 安全位置
      SET     M300  ; 开冲床
      RST     M340  ; 手动冲床1
12508 LD      M300  ; 开冲床
      MPS
      ANDD<=  D8340 D198  ; 右 安全位置
      AND     M600  ; X0-右安全位置
      OUT     M2048  ; 右 安全位
      MPP
      ANDD<=  D8350 D206  ; 左 安全位置
      AND     M605  ; X5-左安全位置
      OUT     M2049  ; 左 安全位
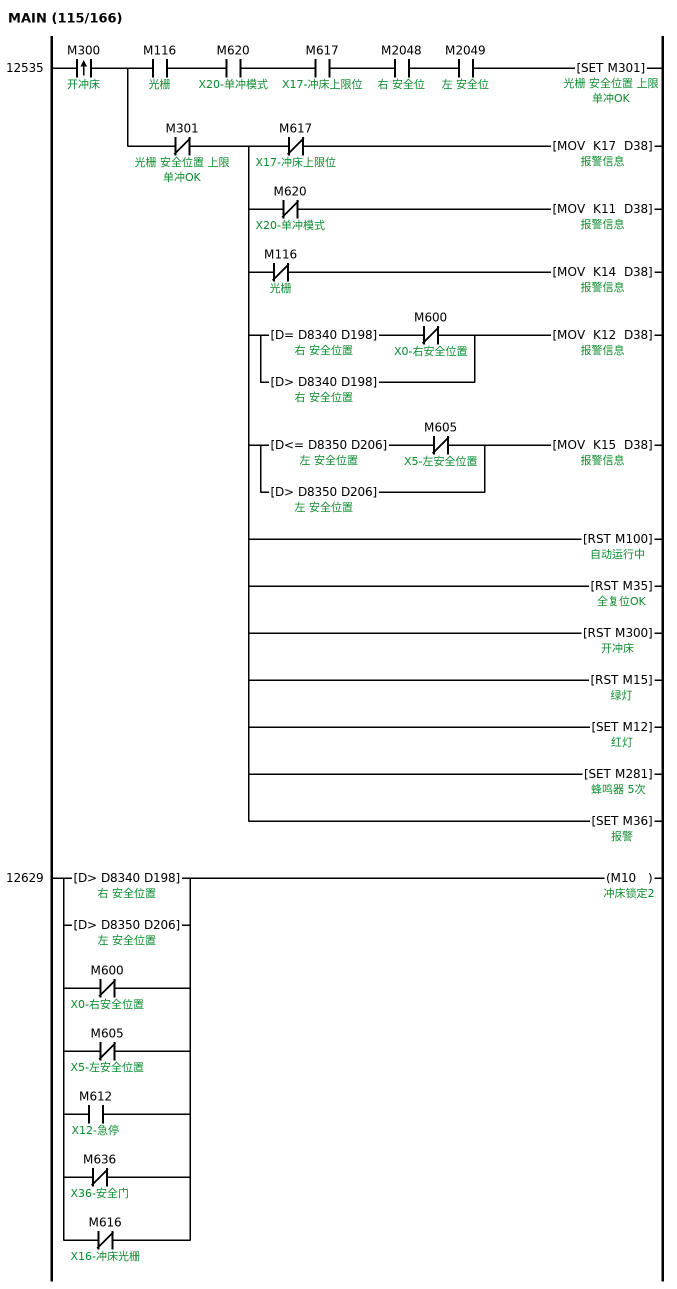
12535 LDP     M300  ; 开冲床
      MPS
      AND     M116  ; 光栅
      AND     M620  ; X20-单冲模式
      AND     M617  ; X17-冲床上限位
      AND     M2048  ; 右 安全位
      AND     M2049  ; 左 安全位
      SET     M301  ; 光栅 安全位置 上限 单冲OK
      MPP
      ANI     M301  ; 光栅 安全位置 上限 单冲OK
      MPS
      ANI     M617  ; X17-冲床上限位
      MOV     K17 D38
      MRD
      ANI     M620  ; X20-单冲模式
      MOV     K11 D38
      MRD
      ANI     M116  ; 光栅
      MOV     K14 D38
      MRD
      LDD=    D8340 D198  ; 右 安全位置
      ANI     M600  ; X0-右安全位置
      ORD>    D8340 D198  ; 右 安全位置
      ANB
      MOV     K12 D38
      MRD
      LDD<=   D8350 D206  ; 左 安全位置
      ANI     M605  ; X5-左安全位置
      ORD>    D8350 D206  ; 左 安全位置
      ANB
      MOV     K15 D38
      MPP
      RST     M100  ; 自动运行中
      RST     M35  ; 全复位OK
      RST     M300  ; 开冲床
      RST     M15  ; 绿灯
      SET     M12  ; 红灯
      SET     M281  ; 蜂鸣器 5次
      SET     M36  ; 报警
12629 LDD>    D8340 D198  ; 右 安全位置
      ORD>    D8350 D206  ; 左 安全位置
      ORI     M600  ; X0-右安全位置
      ORI     M605  ; X5-左安全位置
      OR      M612  ; X12-急停
      ORI     M636  ; X36-安全门
      ORI     M616  ; X16-冲床光栅
      OUT     M10  ; 冲床锁定2
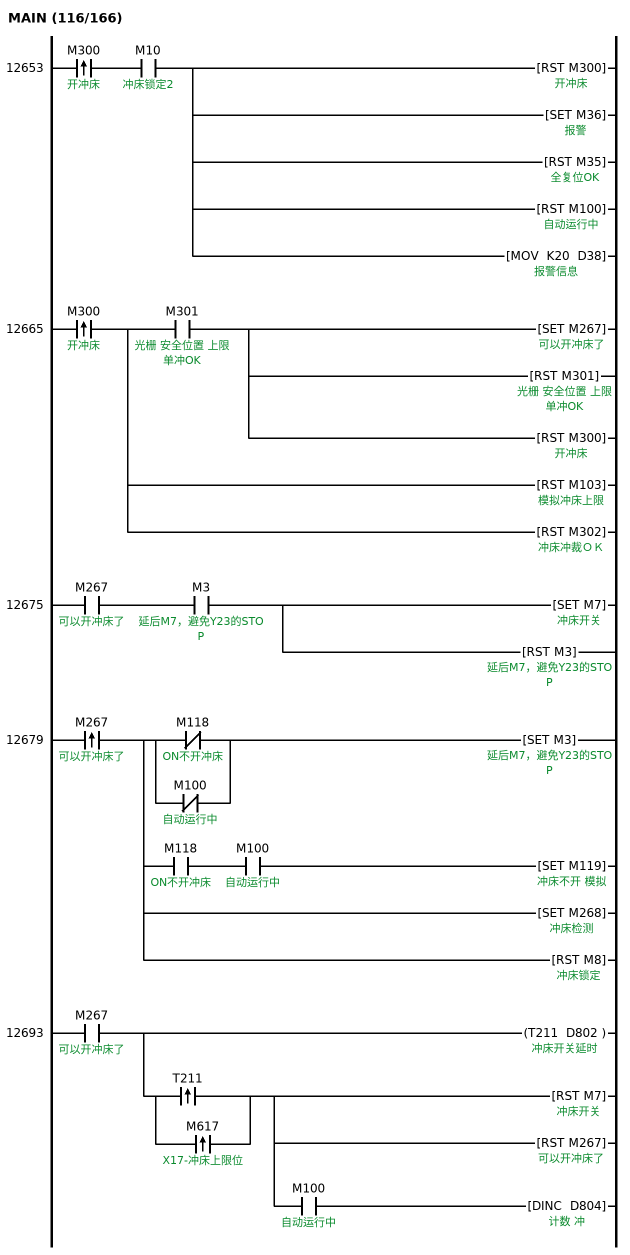
12653 LDP     M300  ; 开冲床
      AND     M10  ; 冲床锁定2
      RST     M300  ; 开冲床
      SET     M36  ; 报警
      RST     M35  ; 全复位OK
      RST     M100  ; 自动运行中
      MOV     K20 D38
12665 LDP     M300  ; 开冲床
      MPS
      AND     M301  ; 光栅 安全位置 上限 单冲OK
      SET     M267  ; 可以开冲床了
      RST     M301  ; 光栅 安全位置 上限 单冲OK
      RST     M300  ; 开冲床
      MPP
      RST     M103  ; 模拟冲床上限
      RST     M302  ; 冲床冲裁ＯＫ
12675 LD      M267  ; 可以开冲床了
      AND     M3  ; 延后M7，避免Y23的STOP
      SET     M7  ; 冲床开关
      RST     M3  ; 延后M7，避免Y23的STOP
12679 LDP     M267  ; 可以开冲床了
      MPS
      LDI     M118  ; ON不开冲床
      ORI     M100  ; 自动运行中
      ANB
      SET     M3  ; 延后M7，避免Y23的STOP
      MRD
      AND     M118  ; ON不开冲床
      AND     M100  ; 自动运行中
      SET     M119  ; 冲床不开 模拟
      MPP
      SET     M268  ; 冲床检测
      RST     M8  ; 冲床锁定
12693 LD      M267  ; 可以开冲床了
      OUT     T211 D802  ; 冲床开关延时
      LDP     T211
      ORP     M617  ; X17-冲床上限位
      ANB
      RST     M7  ; 冲床开关
      RST     M267  ; 可以开冲床了
      AND     M100  ; 自动运行中
      DINC    D804
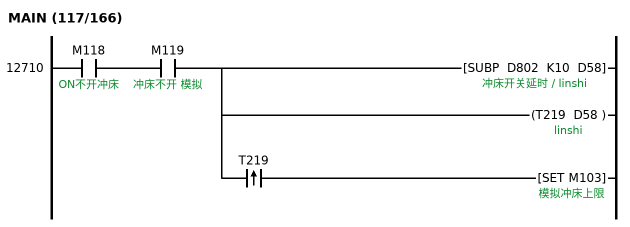
12710 LD      M118  ; ON不开冲床
      AND     M119  ; 冲床不开 模拟
      SUBP    D802 K10 D58  ; linshi
      OUT     T219 D58  ; linshi
      ANDP    T219
      SET     M103  ; 模拟冲床上限
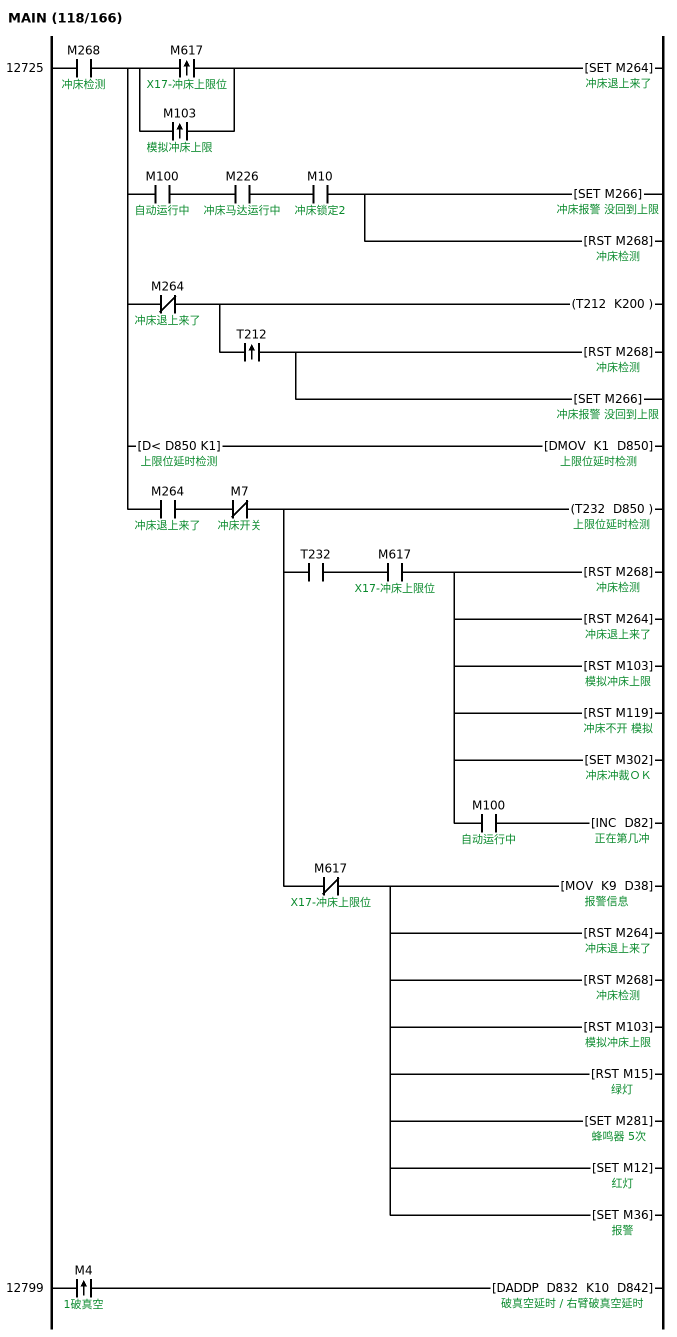
12725 LD      M268  ; 冲床检测
      MPS
      LDP     M617  ; X17-冲床上限位
      ORP     M103  ; 模拟冲床上限
      ANB
      SET     M264  ; 冲床退上来了
      MRD
      AND     M100  ; 自动运行中
      AND     M226  ; 冲床马达运行中
      AND     M10  ; 冲床锁定2
      SET     M266  ; 冲床报警 没回到上限
      RST     M268  ; 冲床检测
      MRD
      ANI     M264  ; 冲床退上来了
      OUT     T212 K200
      ANDP    T212
      RST     M268  ; 冲床检测
      SET     M266  ; 冲床报警 没回到上限
      MRD
      ANDD<   D850 K1  ; 上限位延时检测
      DMOV    K1 D850
      MPP
      AND     M264  ; 冲床退上来了
      ANI     M7  ; 冲床开关
      OUT     T232 D850  ; 上限位延时检测
      MPS
      AND     T232
      AND     M617  ; X17-冲床上限位
      RST     M268  ; 冲床检测
      RST     M264  ; 冲床退上来了
      RST     M103  ; 模拟冲床上限
      RST     M119  ; 冲床不开 模拟
      SET     M302  ; 冲床冲裁ＯＫ
      AND     M100  ; 自动运行中
      INC     D82
      MPP
      ANI     M617  ; X17-冲床上限位
      MOV     K9 D38
      RST     M264  ; 冲床退上来了
      RST     M268  ; 冲床检测
      RST     M103  ; 模拟冲床上限
      RST     M15  ; 绿灯
      SET     M281  ; 蜂鸣器 5次
      SET     M12  ; 红灯
      SET     M36  ; 报警
12799 LDP     M4  ; 1破真空
      DADDP   D832 K10 D842  ; 右臂破真空延时
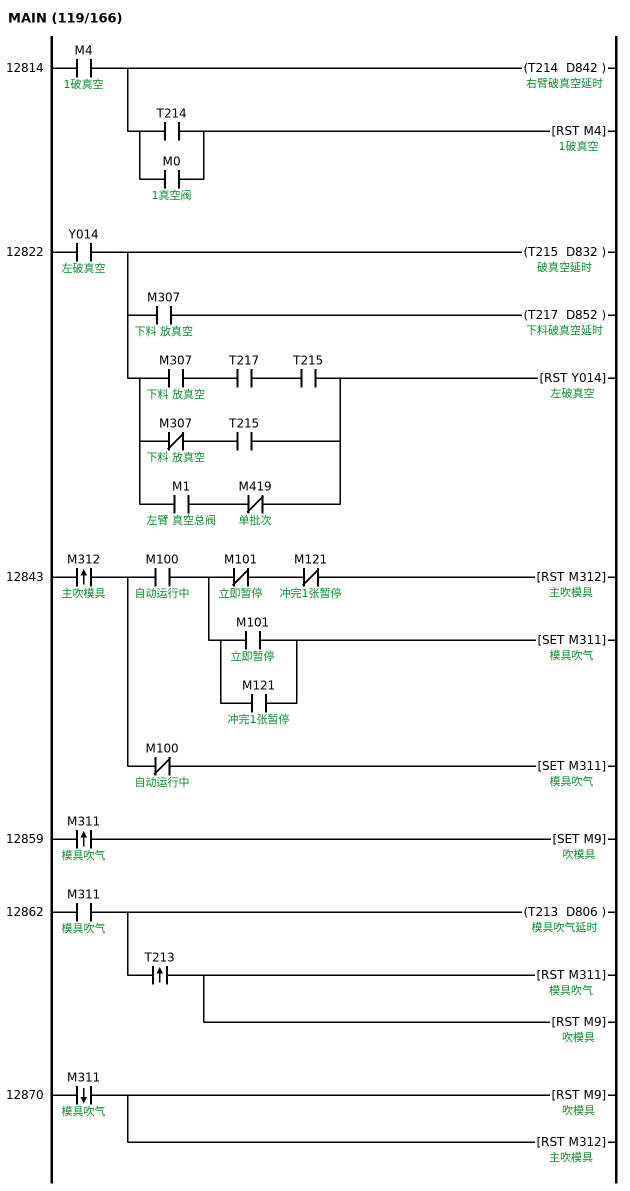
12814 LD      M4  ; 1破真空
      OUT     T214 D842  ; 右臂破真空延时
      LD      T214
      OR      M0  ; 1真空阀
      ANB
      RST     M4  ; 1破真空
12822 LD      Y014  ; 左破真空
      OUT     T215 D832  ; 破真空延时
      MPS
      AND     M307  ; 下料 放真空
      OUT     T217 D852  ; 下料破真空延时
      MPP
      LD      M307  ; 下料 放真空
      AND     T217
      AND     T215
      LDI     M307  ; 下料 放真空
      AND     T215
      ORB
      LD      M1  ; 左臂 真空总阀
      ANI     M419  ; 单批次
      ORB
      ANB
      RST     Y014  ; 左破真空
12843 LDP     M312  ; 主吹模具
      MPS
      AND     M100  ; 自动运行中
      MPS
      ANI     M101  ; 立即暂停
      ANI     M121  ; 冲完1张暂停
      RST     M312  ; 主吹模具
      MPP
      LD      M101  ; 立即暂停
      OR      M121  ; 冲完1张暂停
      ANB
      SET     M311  ; 模具吹气
      MPP
      ANI     M100  ; 自动运行中
      SET     M311  ; 模具吹气
12859 LDP     M311  ; 模具吹气
      SET     M9  ; 吹模具
12862 LD      M311  ; 模具吹气
      OUT     T213 D806  ; 模具吹气延时
      ANDP    T213
      RST     M311  ; 模具吹气
      RST     M9  ; 吹模具
12870 LDF     M311  ; 模具吹气
      RST     M9  ; 吹模具
      RST     M312  ; 主吹模具
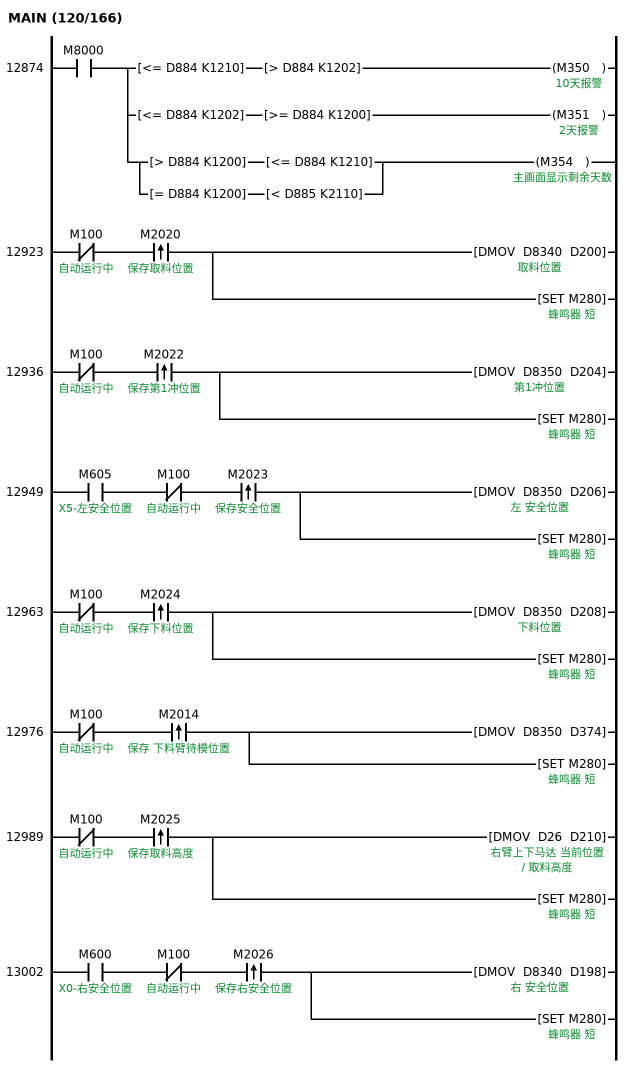
12874 LD      M8000
      MPS
      AND<=   D884 K1210
      AND>    D884 K1202
      OUT     M350  ; 10天报警
      MRD
      AND<=   D884 K1202
      AND>=   D884 K1200
      OUT     M351  ; 2天报警
      MPP
      LD>     D884 K1200
      AND<=   D884 K1210
      LD=     D884 K1200
      AND<    D885 K2110
      ORB
      ANB
      OUT     M354  ; 主画面显示剩余天数
12923 LDI     M100  ; 自动运行中
      ANDP    M2020  ; 保存取料位置
      DMOV    D8340 D200
      SET     M280  ; 蜂鸣器 短
12936 LDI     M100  ; 自动运行中
      ANDP    M2022  ; 保存第1冲位置
      DMOV    D8350 D204
      SET     M280  ; 蜂鸣器 短
12949 LD      M605  ; X5-左安全位置
      ANI     M100  ; 自动运行中
      ANDP    M2023  ; 保存安全位置
      DMOV    D8350 D206
      SET     M280  ; 蜂鸣器 短
12963 LDI     M100  ; 自动运行中
      ANDP    M2024  ; 保存下料位置
      DMOV    D8350 D208
      SET     M280  ; 蜂鸣器 短
12976 LDI     M100  ; 自动运行中
      ANDP    M2014  ; 保存 下料臂待模位置
      DMOV    D8350 D374
      SET     M280  ; 蜂鸣器 短
12989 LDI     M100  ; 自动运行中
      ANDP    M2025  ; 保存取料高度
      DMOV    D26 D210
      SET     M280  ; 蜂鸣器 短
13002 LD      M600  ; X0-右安全位置
      ANI     M100  ; 自动运行中
      ANDP    M2026  ; 保存右安全位置
      DMOV    D8340 D198
      SET     M280  ; 蜂鸣器 短
